DEVICE_TYPE FBRT_WINDOW (* An FBRT device showing a window for HMI *)
  (* Standard: 61499 ITA; Description: Remotely managed windowed device *)
  (* Version 1.0, 2015-11-02, Alois Zoitl, fortiss GmbH, Initial version *)
  VAR_INPUT
    BOUNDS : ARRAY [0..3] OF DINT; (* Initial[x,y,width,height] *)
    GRID : ARRAY [0..1] OF DINT; (* Grid layout[rows,cols] *)
    MGR_ID : WSTRING := "localhost:61499"; (* Device manager socket ID *)
  END_VAR
END_DEVICE_TYPE
